{attribute 'qualified_only'}
{attribute 'to_string'}
TYPE
StationName_e :
(
    Station_105 := 1,
    Station_110 := 2,
    Station_115 := 3,
    Station_120 := 4,
    Station_125 := 5,
    Station_130 := 6,
    Station_135 := 7,
    Station_140 := 8,
    Station_145 := 9,
    Station_150 := 10,
    Station_155 := 11,
    Station_160 := 12,
    Station_165 := 13,
    Station_170 := 14,
    Station_175 := 15,
    Station_176 := 16,
    Station_180 := 17,
    Station_185 := 18
);
END_TYPE

(* stored: Version 1.1.0.1, ProductVersion 3.1.4024.6
   EnumerationTextList StationName_e: Id {9c5c3967-f60b-4d52-bdf8-9d59f2175d7d} *)
